# EPICS substitutions: ek9000App/Db/EL3004.substitutions
file EL3004.template
{       pattern
        {
                TERMINAL,

        }
        {
        }
}
